FUNCTION Queue_FIFO : BOOL
VAR_INPUT
	inputSize : UDINT;
	inputAdr : POINTER TO BYTE;
	
	arrSize : UDINT;
	arrAdr : POINTER TO BYTE;
END_VAR
VAR
END_VAR

FW_MemMove(pDest := arrAdr + inputSize, pSrc := arrAdr, cbLen := arrSize - inputSize);

FW_MemMove(pDest := arrAdr, pSrc := inputAdr, cbLen := inputSize);

END_FUNCTION

(* stored: Version 1.1.0.1, ProductVersion 3.1.4024.9
   POU Queue_FIFO: Id {bba86fe8-a5e4-4329-bde4-32d262471317}, SpecialFunc None *)
